//Batching machine
PROGRAM MAIN
VAR
	vending: Vendingmachine;
	aaa: REAL:= 0;
	bbb: INT:= 3;
	ccc: INT;
	switch: BOOL;
	ntStart:NT_StartProcess;

END_VAR

vending();
UPTIME();

IF switch THEN
	aaa:= aaa + 1;
	switch:= FALSE;
END_IF
ntStart(
	NETID:= , 
	PATHSTR:= 'C:\TwinCAT\3.1\Components\Plc\Tc3PlcHmi\Tc3PlcHmi.exe', 
	DIRNAME:= 'C:\TwinCAT\3.1\Components\Plc\Tc3PlcHmi', 
	COMNDLINE:= , 
	START:= TRUE, 
	TMOUT:= , 
		BUSY=> , 
		ERR=> , 
	ERRID=> );

END_PROGRAM

(* stored: Version 1.1.0.1, ProductVersion 3.1.4024.10
   POU MAIN: Id {c4f4d626-e859-4cd7-af51-566a5ab15381}, SpecialFunc None *)
